FUNCTION_BLOCK FB_Unit
VAR_INPUT
	OpMode: E_OpMode;
END_VAR
VAR_OUTPUT
END_VAR
VAR
END_VAR

END_FUNCTION_BLOCK

(* stored: Version 1.1.0.1, ProductVersion 3.1.4024.11
   POU FB_Unit: Id {ab8dbb11-5f04-4f82-9f6d-1cfe55ae9701}, SpecialFunc None *)
